FUNCTION_BLOCK Canal_UV (* Composite Function Block Type *)
  (* Standard: 61499-2 *)
  (* Version 0.0, 03/03/2026, template *)
  PACKAGE Hidryco.HidrycoLib;
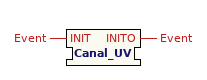
  EVENT_INPUT
    INIT;
  END_EVENT
  EVENT_OUTPUT
    INITO;
  END_EVENT
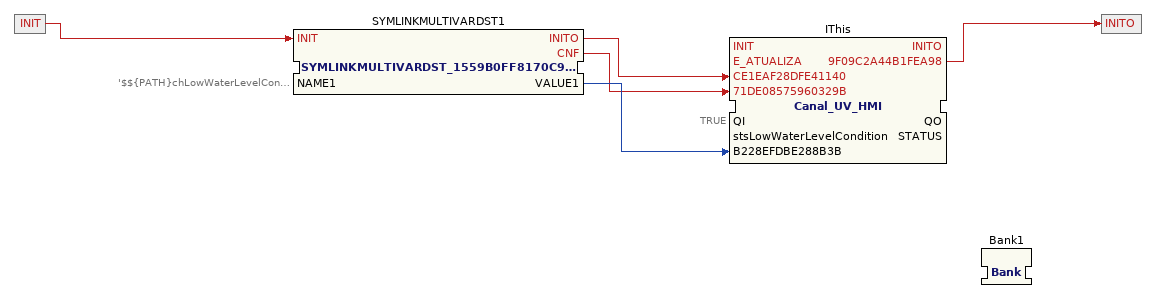
  FBS
    SYMLINKMULTIVARDST1 : SYMLINKMULTIVARDST_1559B0FF8170C9BA0(NAME1 := '$${PATH}chLowWaterLevelCondition'); {SET_ATTRIBUTE(Configuration.GenericFBType.InterfaceParams, Runtime.System#I:=1;VALUE${I$}:BOOL)}
    Bank1 : Bank;
    IThis : Canal_UV_HMI(QI := TRUE);
  END_FBS
  EVENT_CONNECTIONS
    INIT TO SYMLINKMULTIVARDST1.INIT;
    SYMLINKMULTIVARDST1.INITO TO IThis.CE1EAF28DFE41140;
    SYMLINKMULTIVARDST1.CNF TO IThis.71DE08575960329B;
    IThis.9F09C2A44B1FEA98 TO INITO;
  END_CONNECTIONS
  DATA_CONNECTIONS
    SYMLINKMULTIVARDST1.VALUE1 TO IThis.B228EFDBE288B3B;
  END_CONNECTIONS
END_FUNCTION_BLOCK
